// Mitsubishi GX Works2 project: LRI - PLC - AULA 11.1   PLC: Q03UDV

// task Task_01 (event TRUE, interval 0, priority 31): POU_01

PROGRAM POU_01
VAR
  iDR : ARRAY [0..9] OF INT;
  stOperacoes_1 : stOperacoes;
  stOperacoes_2 : stOperacoes;
  stOperacoes_3 : stOperacoes;
  stOperacoes_4 : stOperacoes;
  tester : INT;
  stOperacoes_5 : stOperacoes;
END_VAR


iDR[0] := stSoma( 100 , 500 );

iDR[1] := stSubtracao( 100 , 500 );


iDR[2] := stMultiplica( 100 , 500 );

iDR[3] := stDivisao( 100 , 500 );

stOperacoes_2(i_VarUmOperacao:= 100 ,i_VarDoisOperacao:= 200 ); (*,o_VarSomaSt:= 100,o_VarSubtracaoSt:= 200  ,o_VarMultiplicaoSt:= 100 ,
	o_VarDivisaoSt:= 200  );*)
	
tester:= stOperacoes_2.o_VarSomaSt;

stOperacoes_5(i_VarUmOperacao:= 100 ,i_VarDoisOperacao:= 200 ,o_VarSomaSt:= iDR[4] ,o_VarSubtracaoSt:= iDR[5] ,o_VarMultiplicaoSt:= iDR[5] ,
	o_VarDivisaoSt:= iDR[6] );
END_PROGRAM

FUNCTION stSoma
VAR_INPUT
  i_VarDoisSoma : INT;
  i_VarUmSoma : INT;
END_VAR


stSoma := i_VarUmSoma + i_VarDoisSoma;
END_FUNCTION

FUNCTION stSubtracao
VAR_INPUT
  i_VarUmSubtracao : INT;
  i_VarDoisSubtracao : INT;
END_VAR
stSubtracao := i_VarUmSubtracao - i_VarDoisSubtracao;
END_FUNCTION

FUNCTION stMultiplica
VAR_INPUT
  i_VarUmMultiplicar : INT;
  i_VarDoisMultiplicar : INT;
END_VAR


stMultiplica := i_VarUmMultiplicar * i_VarDoisMultiplicar;
END_FUNCTION

FUNCTION stDivisao
VAR_INPUT
  i_VarUmDivisao : INT;
  i_VarDoisDivisao : INT;
END_VAR
stDivisao := i_VarUmDivisao MOD i_VarDoisDivisao;
END_FUNCTION

FUNCTION_BLOCK stOperacoes
VAR_INPUT
  i_VarUmOperacao : INT;
  i_VarDoisOperacao : INT;
END_VAR
VAR_OUTPUT
  o_VarSomaSt : INT;
  o_VarSubtracaoSt : INT;
  o_VarMultiplicaoSt : INT;
  o_VarDivisaoSt : INT;
END_VAR


o_VarSomaSt := stSoma( i_VarUmOperacao, i_VarDoisOperacao);

o_VarSubtracaoSt := stSubtracao( i_VarUmOperacao, i_VarDoisOperacao);

o_VarMultiplicaoSt := stMultiplica( i_VarUmOperacao, i_VarDoisOperacao);


o_VarDivisaoSt := stDivisao( i_VarUmOperacao, i_VarDoisOperacao);
END_FUNCTION_BLOCK
